# EPICS StreamDevice protocol: measm905Sup/measm905.proto
Terminator = CR;
ReplyTimeout = 2000;

getCurrPressure {
    out "*01D"; #Over ASCII Protocol, request reading
    in "%d"; #The Pressure reading
}
